PROGRAM MAIN
VAR
	ConveyorTracking01		: 	ConveyorTracking;	
	ConveyorTracking02		: 	ConveyorTracking;
	ConveyorTracking03		: 	ConveyorTracking;
	EncoderResolution		:	REAL:=0.2;
	TrackingAccuracy		:	REAL:=1.0;
	Reset					: 	BOOL;
	tpDrvStop				: 	TP;
	DroppedProducts1		:	CTU;
	DroppedProducts2		:	CTU;
	DroppedProducts3		:	CTU;
END_VAR

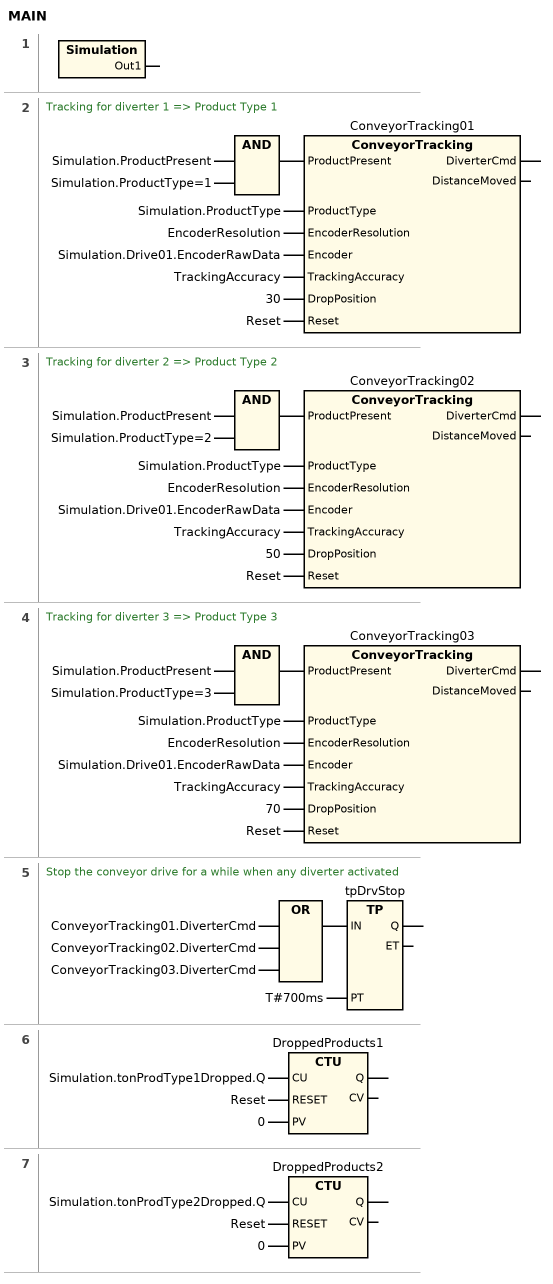
// NETWORK 1
Simulation();

// NETWORK 2
// Tracking for diverter 1 => Product Type 1
ConveyorTracking01(
    ProductPresent := Simulation.ProductPresent AND (Simulation.ProductType=1),
    ProductType := Simulation.ProductType,
    EncoderResolution := EncoderResolution,
    Encoder := Simulation.Drive01.EncoderRawData,
    TrackingAccuracy := TrackingAccuracy,
    DropPosition := 30,
    Reset := Reset); // ConveyorTracking

// NETWORK 3
// Tracking for diverter 2 => Product Type 2
ConveyorTracking02(
    ProductPresent := Simulation.ProductPresent AND (Simulation.ProductType=2),
    ProductType := Simulation.ProductType,
    EncoderResolution := EncoderResolution,
    Encoder := Simulation.Drive01.EncoderRawData,
    TrackingAccuracy := TrackingAccuracy,
    DropPosition := 50,
    Reset := Reset); // ConveyorTracking

// NETWORK 4
// Tracking for diverter 3 => Product Type 3
ConveyorTracking03(
    ProductPresent := Simulation.ProductPresent AND (Simulation.ProductType=3),
    ProductType := Simulation.ProductType,
    EncoderResolution := EncoderResolution,
    Encoder := Simulation.Drive01.EncoderRawData,
    TrackingAccuracy := TrackingAccuracy,
    DropPosition := 70,
    Reset := Reset); // ConveyorTracking

// NETWORK 5
// Stop the conveyor drive for a while when any diverter activated
tpDrvStop(IN := ConveyorTracking01.DiverterCmd OR ConveyorTracking02.DiverterCmd OR ConveyorTracking03.DiverterCmd, PT := T#700ms); // TP

// NETWORK 6
DroppedProducts1(CU := Simulation.tonProdType1Dropped.Q, RESET := Reset, PV := 0); // CTU

// NETWORK 7
DroppedProducts2(CU := Simulation.tonProdType2Dropped.Q, RESET := Reset, PV := 0); // CTU

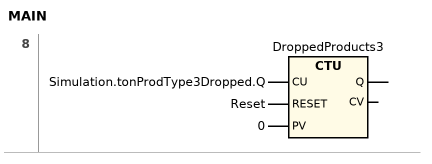
// NETWORK 8
DroppedProducts3(CU := Simulation.tonProdType3Dropped.Q, RESET := Reset, PV := 0); // CTU

END_PROGRAM

(* stored: Version 1.1.0.1, ProductVersion 3.1.4024.15
   POU MAIN: Id {c841af35-eae6-445e-8aa9-1035a2ad2f08}, SpecialFunc None *)
